INTERFACE PUBLIC I_JogMoveBuilder EXTENDS __System.IQueryInterface

METHOD PUBLIC Acceleration : I_MoveBuilder
VAR_INPUT
	value : LREAL;
END_VAR
END_METHOD

METHOD PUBLIC BuildBackwardsCommand : I_MoveCommand
END_METHOD

METHOD PUBLIC BuildForwardCommand : I_MoveCommand
END_METHOD

METHOD PUBLIC Deceleration : I_MoveBuilder
VAR_INPUT
	value : LREAL;
END_VAR
END_METHOD

METHOD PUBLIC Distance : I_JogMoveBuilder
VAR_INPUT
	value : LREAL;
END_VAR
END_METHOD

METHOD PUBLIC Jerk : I_MoveBuilder
VAR_INPUT
	value : LREAL;
END_VAR
END_METHOD

METHOD PUBLIC Velocity : I_MoveBuilder
VAR_INPUT
	value : LREAL;
END_VAR
END_METHOD

END_INTERFACE

(* stored: Version 1.1.0.1, ProductVersion 3.1.4024.12
   Itf I_JogMoveBuilder: Id {63011fe5-43c5-0691-2811-26343292cc88}
   Method Acceleration: Id {af89edba-a005-0f7a-08ee-62427ab92e8c}
   Method BuildBackwardsCommand: Id {811b0cdc-1229-0e51-31b7-d139d434f5da}
   Method BuildForwardCommand: Id {eb48d50f-4383-072c-36b0-a8587d3e78d1}
   Method Deceleration: Id {81f51863-dcaa-08e1-131a-d2d14e3869a9}
   Method Distance: Id {e48b5c47-c8ce-0805-3136-ccdb4eb1e486}
   Method Jerk: Id {515fb89c-e14f-0eca-3e64-4213131f22cc}
   Method Velocity: Id {e754fcf6-ed62-04aa-1e93-2f61470560c8} *)
